{attribute addProperty BoxType "EJ3318-0000-0017"}
{attribute addProperty Id "StatusAT %I*Status_C3A5DD7C1621ValueAT %I*INT16217"}
{attribute addProperty CRC "397281499"}
{attribute addProperty SizeInBites "32"}
{attribute addProperty SizeInBytes "4"}
TYPE TC_Channel_17AE08DB :
STRUCT
	{attribute addProperty Name "Status"}
	Status AT %I* : Status_C3A5DD7C;
	{attribute addProperty Name "Value"}
	Value AT %I* : INT;
END_STRUCT
END_TYPE

(* stored: Version 1.2.0.0, ProductVersion 3.1.4024.9
   DUT TC_Channel_17AE08DB: Id {74bde96a-76c1-499a-869c-3ba166699e3e} *)
